SUBAPPLICATION Uebung_010b7_AX (* Toggle Flip-Flop mit IE Button_A1 BT_RELEASED_UNLATCHED *)
  (* Standard: 61499-2; Description: Copyright (c) 2023 Meisterschulen am Ostbahnhof This program and the accompanying materials are made available under the terms of the Eclipse Public License 2.0 which is available at https://www.eclipse.org/legal/epl-2.0/ SPDX-License-Identifier: EPL-2.0 *)
  (* Version 1.0, 2026-01-15, Franz Höpfinger, Meisterschulen am Ostbahnhof, initial API and implementation and/or initial documentation *)
  PACKAGE Uebungen;
  IMPORT Uebungen::const::UT::DefaultPool::Button_A1;
  IMPORT isobus::UT::io::Button::ButtonActivationCode::BT_RELEASED_UNLATCHED;
  IMPORT logiBUS::io::DQ::logiBUS_DO::Output_Q1;
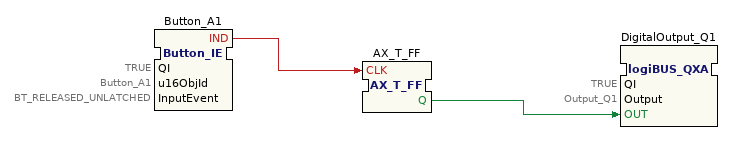
  FBS
    DigitalOutput_Q1 : logiBUS::io::DQ::logiBUS_QXA(QI := TRUE, Output := Output_Q1);
    Button_A1 : isobus::UT::io::Button::Button_IE(QI := TRUE, u16ObjId := Button_A1, InputEvent := BT_RELEASED_UNLATCHED);
    AX_T_FF : adapter::events::unidirectional::AX_T_FF;
  END_FBS
  EVENT_CONNECTIONS
    Button_A1.IND TO AX_T_FF.CLK;
  END_CONNECTIONS
  ADAPTER_CONNECTIONS
    AX_T_FF.Q TO DigitalOutput_Q1.OUT;
  END_CONNECTIONS
END_SUBAPPLICATION
